{attribute 'GeneratedUsingTerminal: EL5101-0000-1019'}
{attribute addProperty BoxType "EL5101-0000-1019"}
{attribute addProperty Id "ENC_Status_compactAT %I*ENC_Status_compact_D1AA753920ENC_Control_compactAT %Q*ENC_Control_compact_6FDDC6696WcStateAT %I*WcState_9091E0EB2InfoDataAT %I*InfoData_94A18F5E2"}
{attribute addProperty CRC "567717468"}
{attribute addProperty Size "30"}
TYPE EL5101_21D6AE5C EXTENDS EtcSlaveTerminalBase_947E5A46 :
STRUCT
	{attribute addProperty Name "ENC_Status_compact"}
	ENC_Status_compact : ENC_Status_compact_D1AA7539;
	{attribute addProperty Name "ENC_Control_compact"}
	ENC_Control_compact : ENC_Control_compact_6FDDC669;
	{attribute addProperty Name "WcState"}
	WcState : WcState_9091E0EB;
	{attribute addProperty Name "InfoData"}
	InfoData : InfoData_94A18F5E;
END_STRUCT
END_TYPE

(* stored: Version 1.2.0.0, ProductVersion 3.1.4024.9
   DUT EL5101_21D6AE5C: Id {70052d2c-ec33-4226-886e-718580e38e15} *)
